SYSTEM TRAFFIC_Distributed (* System Configuration *)
  (* Standard: 61499-1 *)
  (* Version 0.4, 2009-03-05, JHC, Holobloc Inc., Deleted Application. *)
  (* Version 0.3, 2003-12-05, JHC, Rockwell Automation, Renamed from NEWSYSTEM. *)
  (* Version 0.2, 2002-11-05, JHC, Rockwell Automation, Fixed missing (empty) FBD in Application. *)
  (* Version 0.1, 2002-01-17, JHC, Rockwell Automation, Minor cleanup *)
  (* Version 0.0, 2000-05-27, JHC, Rockwell Automation *)
  DEVICE Device1 : FRAME_DEVICE(BOUNDS := [400,100,200,200], GRID := [1])
    RESOURCE View : PANEL_RESOURCE(ROWS := 6, COLS := 1)
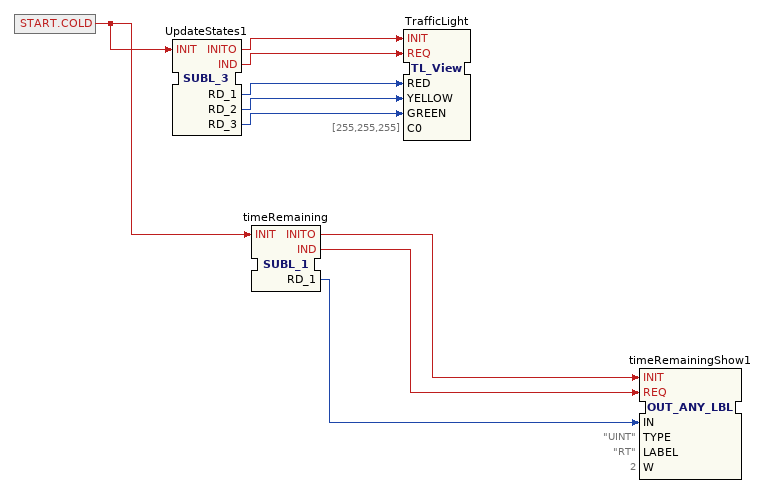
      FBS
        TrafficLight : TL_View(C0 := [255,255,255]);
        UpdateStates1 : SUBL_3;
        timeRemaining : SUBL_1;
        timeRemainingShow1 : OUT_ANY_LBL(TYPE := "UINT", LABEL := "RT", W := 2);
      END_FBS
      EVENT_CONNECTIONS
        START.COLD TO UpdateStates1.INIT;
        UpdateStates1.INITO TO TrafficLight.INIT;
        UpdateStates1.IND TO TrafficLight.REQ;
        START.COLD TO timeRemaining.INIT;
        timeRemaining.INITO TO timeRemainingShow1.INIT;
        timeRemaining.IND TO timeRemainingShow1.REQ;
      END_CONNECTIONS
      DATA_CONNECTIONS
        UpdateStates1.RD_1 TO TrafficLight.RED;
        UpdateStates1.RD_2 TO TrafficLight.YELLOW;
        UpdateStates1.RD_3 TO TrafficLight.GREEN;
        timeRemaining.RD_1 TO timeRemainingShow1.IN;
      END_CONNECTIONS
    END_RESOURCE
    RESOURCE HMI : PANEL_RESOURCE(ROWS := 6, COLS := 1)
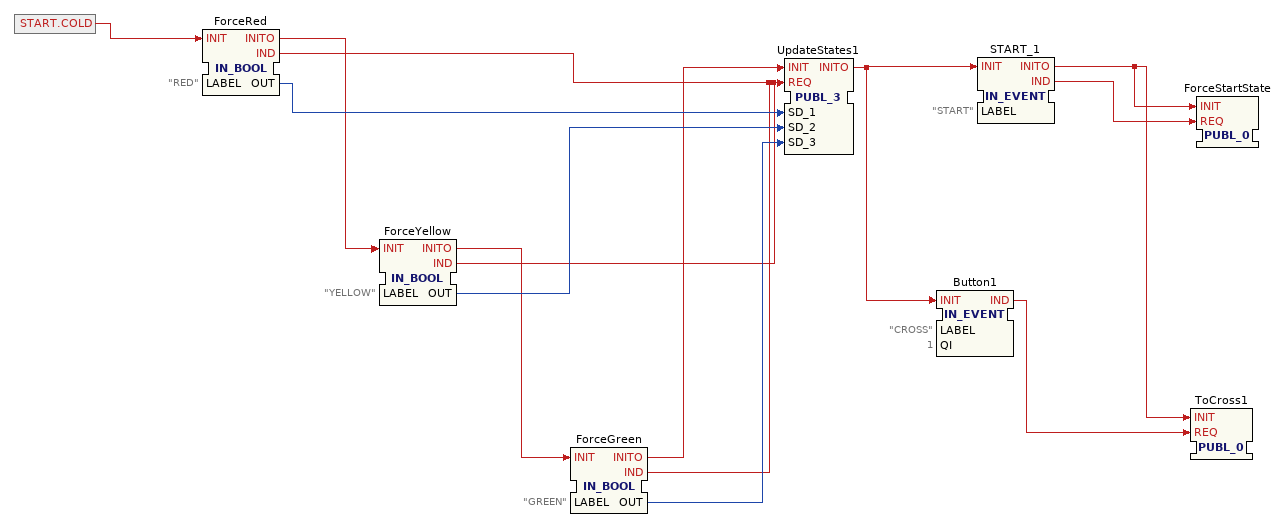
      FBS
        ForceRed : IN_BOOL(LABEL := "RED");
        UpdateStates1 : PUBL_3;
        ForceYellow : IN_BOOL(LABEL := "YELLOW");
        ForceGreen : IN_BOOL(LABEL := "GREEN");
        START_1 : IN_EVENT(LABEL := "START");
        ForceStartState : PUBL_0;
        Button1 : IN_EVENT(LABEL := "CROSS", QI := 1);
        ToCross1 : PUBL_0;
      END_FBS
      EVENT_CONNECTIONS
        START.COLD TO ForceRed.INIT;
        ForceRed.INITO TO ForceYellow.INIT;
        ForceYellow.INITO TO ForceGreen.INIT;
        ForceGreen.INITO TO UpdateStates1.INIT;
        ForceRed.IND TO UpdateStates1.REQ;
        ForceYellow.IND TO UpdateStates1.REQ;
        ForceGreen.IND TO UpdateStates1.REQ;
        UpdateStates1.INITO TO START_1.INIT;
        START_1.INITO TO ForceStartState.INIT;
        START_1.IND TO ForceStartState.REQ;
        UpdateStates1.INITO TO Button1.INIT;
        START_1.INITO TO ToCross1.INIT;
        Button1.IND TO ToCross1.REQ;
      END_CONNECTIONS
      DATA_CONNECTIONS
        ForceRed.OUT TO UpdateStates1.SD_1;
        ForceYellow.OUT TO UpdateStates1.SD_2;
        ForceGreen.OUT TO UpdateStates1.SD_3;
      END_CONNECTIONS
    END_RESOURCE
    RESOURCE Control : EMB_RES
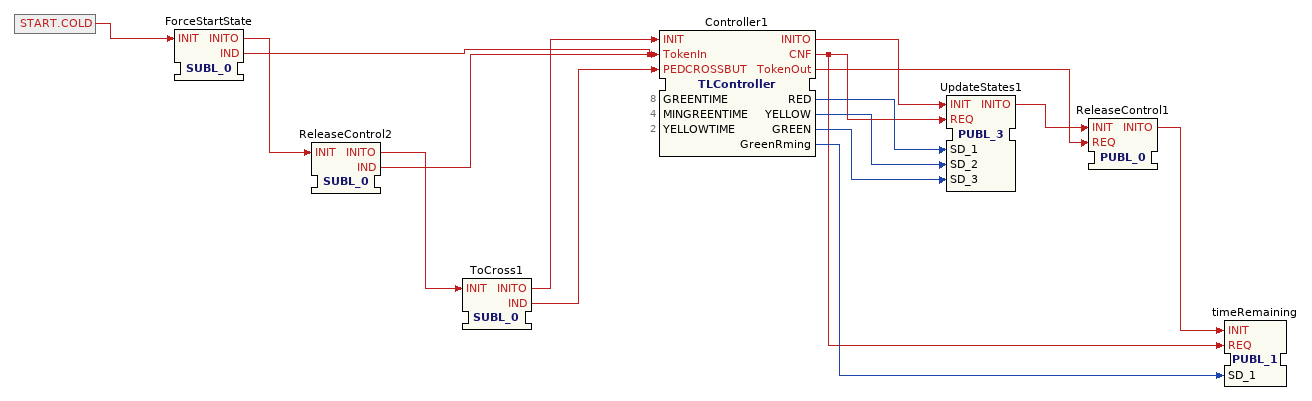
      FBS
        ForceStartState : SUBL_0;
        ReleaseControl2 : SUBL_0;
        ToCross1 : SUBL_0;
        Controller1 : TLController(GREENTIME := 8, MINGREENTIME := 4, YELLOWTIME := 2);
        UpdateStates1 : PUBL_3;
        ReleaseControl1 : PUBL_0;
        timeRemaining : PUBL_1;
      END_FBS
      EVENT_CONNECTIONS
        START.COLD TO ForceStartState.INIT;
        ForceStartState.INITO TO ReleaseControl2.INIT;
        ReleaseControl2.INITO TO ToCross1.INIT;
        ToCross1.INITO TO Controller1.INIT;
        ReleaseControl2.IND TO Controller1.TokenIn;
        ToCross1.IND TO Controller1.PEDCROSSBUT;
        ForceStartState.IND TO Controller1.TokenIn;
        Controller1.INITO TO UpdateStates1.INIT;
        UpdateStates1.INITO TO ReleaseControl1.INIT;
        ReleaseControl1.INITO TO timeRemaining.INIT;
        Controller1.CNF TO UpdateStates1.REQ;
        Controller1.CNF TO timeRemaining.REQ;
        Controller1.TokenOut TO ReleaseControl1.REQ;
      END_CONNECTIONS
      DATA_CONNECTIONS
        Controller1.RED TO UpdateStates1.SD_1;
        Controller1.YELLOW TO UpdateStates1.SD_2;
        Controller1.GREEN TO UpdateStates1.SD_3;
        Controller1.GreenRming TO timeRemaining.SD_1;
      END_CONNECTIONS
    END_RESOURCE
    RESOURCE Model : EMB_RES
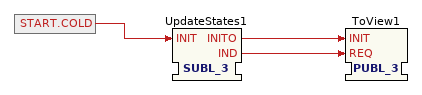
      FBS
        UpdateStates1 : SUBL_3;
        ToView1 : PUBL_3;
      END_FBS
      EVENT_CONNECTIONS
        UpdateStates1.INITO TO ToView1.INIT;
        UpdateStates1.IND TO ToView1.REQ;
        START.COLD TO UpdateStates1.INIT;
      END_CONNECTIONS
    END_RESOURCE
  END_DEVICE
  DEVICE Device2 : FRAME_DEVICE(BOUNDS := [600,100,200,200], GRID := [1])
    RESOURCE View : PANEL_RESOURCE(ROWS := 6, COLS := 1)
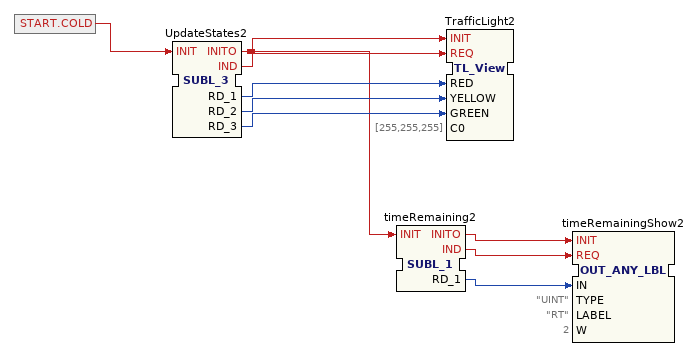
      FBS
        TrafficLight2 : TL_View(C0 := [255,255,255]);
        UpdateStates2 : SUBL_3;
        timeRemaining2 : SUBL_1;
        timeRemainingShow2 : OUT_ANY_LBL(TYPE := "UINT", LABEL := "RT", W := 2);
      END_FBS
      EVENT_CONNECTIONS
        START.COLD TO UpdateStates2.INIT;
        UpdateStates2.INITO TO TrafficLight2.INIT;
        UpdateStates2.IND TO TrafficLight2.REQ;
        UpdateStates2.INITO TO timeRemaining2.INIT;
        timeRemaining2.INITO TO timeRemainingShow2.INIT;
        timeRemaining2.IND TO timeRemainingShow2.REQ;
      END_CONNECTIONS
      DATA_CONNECTIONS
        UpdateStates2.RD_1 TO TrafficLight2.RED;
        UpdateStates2.RD_2 TO TrafficLight2.YELLOW;
        UpdateStates2.RD_3 TO TrafficLight2.GREEN;
        timeRemaining2.RD_1 TO timeRemainingShow2.IN;
      END_CONNECTIONS
    END_RESOURCE
    RESOURCE Control : EMB_RES
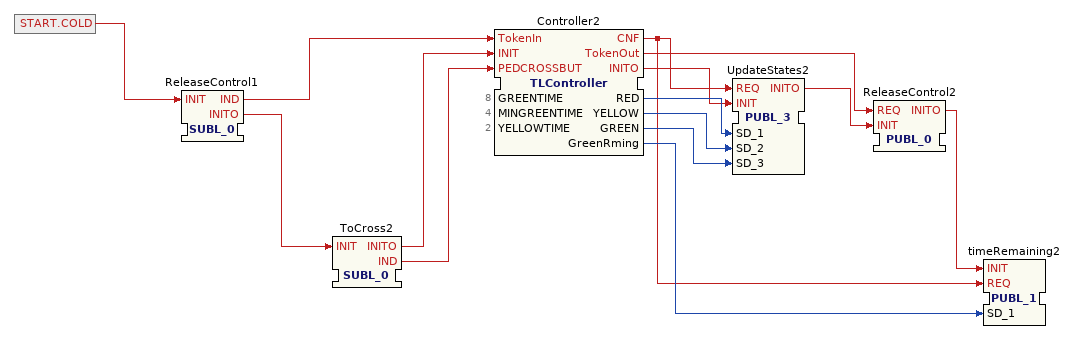
      FBS
        ReleaseControl1 : SUBL_0;
        ToCross2 : SUBL_0;
        Controller2 : TLController(GREENTIME := 8, MINGREENTIME := 4, YELLOWTIME := 2);
        UpdateStates2 : PUBL_3;
        ReleaseControl2 : PUBL_0;
        timeRemaining2 : PUBL_1;
      END_FBS
      EVENT_CONNECTIONS
        Controller2.CNF TO UpdateStates2.REQ;
        Controller2.TokenOut TO ReleaseControl2.REQ;
        START.COLD TO ReleaseControl1.INIT;
        ReleaseControl1.IND TO Controller2.TokenIn;
        ReleaseControl1.INITO TO ToCross2.INIT;
        ToCross2.INITO TO Controller2.INIT;
        ToCross2.IND TO Controller2.PEDCROSSBUT;
        Controller2.INITO TO UpdateStates2.INIT;
        UpdateStates2.INITO TO ReleaseControl2.INIT;
        ReleaseControl2.INITO TO timeRemaining2.INIT;
        Controller2.CNF TO timeRemaining2.REQ;
      END_CONNECTIONS
      DATA_CONNECTIONS
        Controller2.RED TO UpdateStates2.SD_1;
        Controller2.YELLOW TO UpdateStates2.SD_2;
        Controller2.GREEN TO UpdateStates2.SD_3;
        Controller2.GreenRming TO timeRemaining2.SD_1;
      END_CONNECTIONS
    END_RESOURCE
    RESOURCE HMI : PANEL_RESOURCE(ROWS := 6, COLS := 1)
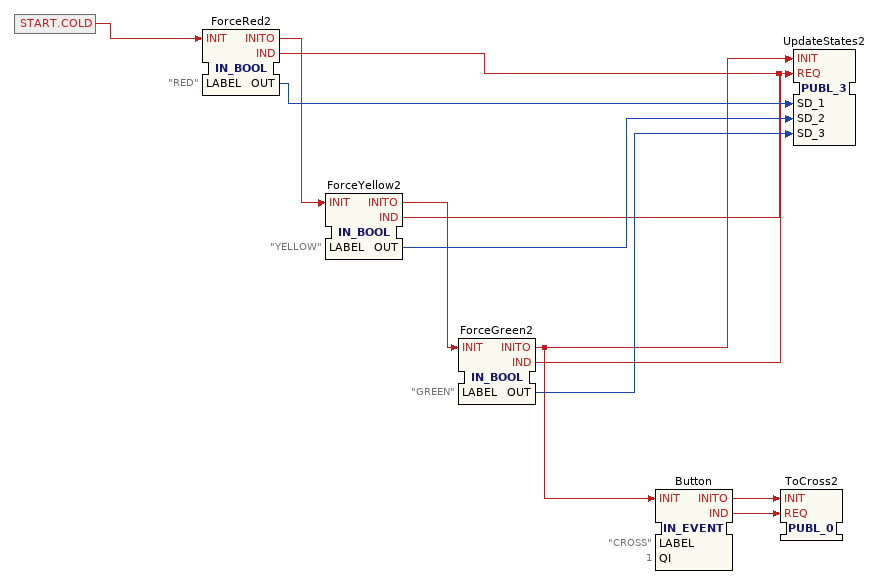
      FBS
        ForceRed2 : IN_BOOL(LABEL := "RED");
        UpdateStates2 : PUBL_3;
        ForceYellow2 : IN_BOOL(LABEL := "YELLOW");
        ForceGreen2 : IN_BOOL(LABEL := "GREEN");
        Button : IN_EVENT(LABEL := "CROSS", QI := 1);
        ToCross2 : PUBL_0;
      END_FBS
      EVENT_CONNECTIONS
        START.COLD TO ForceRed2.INIT;
        ForceRed2.INITO TO ForceYellow2.INIT;
        ForceYellow2.INITO TO ForceGreen2.INIT;
        ForceGreen2.INITO TO UpdateStates2.INIT;
        ForceRed2.IND TO UpdateStates2.REQ;
        ForceYellow2.IND TO UpdateStates2.REQ;
        ForceGreen2.IND TO UpdateStates2.REQ;
        ForceGreen2.INITO TO Button.INIT;
        Button.INITO TO ToCross2.INIT;
        Button.IND TO ToCross2.REQ;
      END_CONNECTIONS
      DATA_CONNECTIONS
        ForceRed2.OUT TO UpdateStates2.SD_1;
        ForceYellow2.OUT TO UpdateStates2.SD_2;
        ForceGreen2.OUT TO UpdateStates2.SD_3;
      END_CONNECTIONS
    END_RESOURCE
    RESOURCE Model : EMB_RES
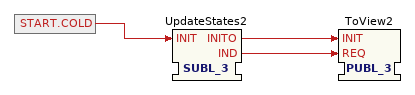
      FBS
        UpdateStates2 : SUBL_3;
        ToView2 : PUBL_3;
      END_FBS
      EVENT_CONNECTIONS
        UpdateStates2.INITO TO ToView2.INIT;
        UpdateStates2.IND TO ToView2.REQ;
        START.COLD TO UpdateStates2.INIT;
      END_CONNECTIONS
    END_RESOURCE
  END_DEVICE
END_SYSTEM
